TYPE ST_HalfAuto_Status :
STRUCT
END_STRUCT
END_TYPE

(* stored: Version 1.1.0.1, ProductVersion 3.1.4024.13
   DUT ST_HalfAuto_Status: Id {78e08219-fc5f-415d-b5e5-568ca5b5a479} *)
